// TwinCAT 3 PLC project Untitled1
// ProgramVersion: 3.1.4023.0
// libraries:
//   Tc2_Standard, * (Beckhoff Automation GmbH)
//   Tc2_System, * (Beckhoff Automation GmbH)
//   Tc3_Module, * (Beckhoff Automation GmbH)
// project tree:
//   / PlcTask.TcTTO
//   POUs/ fb_add.TcPOU, MAIN.TcPOU
// real-time tasks:
//   TASK PlcTask: cycle T#10ms, priority 20, ADS port 350

CONFIGURATION Untitled1
    RESOURCE PLC ON TwinCAT3
        TASK PlcTask(INTERVAL := T#10ms, PRIORITY := 20);
        PROGRAM MAIN WITH PlcTask : MAIN;
    END_RESOURCE
END_CONFIGURATION

// ---- POUs/MAIN.TcPOU
PROGRAM MAIN
VAR
	a:INT;
	b:INT;
	c:INT;
	
	enable: BOOL;
	
	
	fbadd1:fb_add;
	
	cc: INT;
END_VAR


IF enable THEN
	c:=a+b;
ELSE
	c:=0;
END_IF

fbadd1(in1:=a , in2:=b , out=> cc);

END_PROGRAM

// ---- POUs/fb_add.TcPOU
FUNCTION_BLOCK fb_add
VAR_INPUT
	in1:INT;
	in2:INT;
END_VAR
VAR_OUTPUT
	out:INT;
	
END_VAR
VAR
END_VAR


out :=in1+in2;

END_FUNCTION_BLOCK
